// TIA Portal project "TestCase4_S1200_Zonder_Fouten " (V18)

(* hardware
DEVICE "S7-1200 station_1"  S7-1200 Station
   slot 0: "Rack_0"  S7-1200 Rack  Rack  V1.0
   slot 1: "PLC_1"  CPU 1212C DC/DC/DC  6ES7 212-1AE40-0XB0  V4.6
*)

// ===== PLC "PLC_1"  CPU 1212C DC/DC/DC =====

VAR_GLOBAL   // PLC tag table "Default tag table"
   "sensor1" AT %I0.0 : Bool;
   "lampA" AT %Q0.0 : Bool;
   "lampB" AT %Q0.1 : Bool;
   "Tag_1" AT %M101.0 : Bool;
   "Tag_2" AT %M100.0 : Bool;
   "Tag_4" AT %M100.1 : Bool;
   "Tag_5" AT %M100.2 : Bool;
   "sensor2" AT %I0.1 : Bool;
   "sensor3" AT %I0.2 : Bool;
   "Tag_6" AT %M103.0 : Bool;
   "Tag_7" AT %M102.0 : Bool;
END_VAR

DATA_BLOCK "Data_block_1"   // DB1
{ S7_Optimized_Access := 'FALSE' }
VERSION : 0.1
   VAR
      sensor1 : Bool;
      sensor2 : Bool;
      sensor3 : Bool;
   END_VAR
BEGIN
END_DATA_BLOCK

DATA_BLOCK "Data_block_2"   // DB2
{ S7_Optimized_Access := 'FALSE' }
VERSION : 0.1
   VAR
      lampA : Bool;
      lampB : Bool;
   END_VAR
BEGIN
END_DATA_BLOCK

FUNCTION "State0" : Void   // FC1, FBD
{ S7_Optimized_Access := 'TRUE' }
VERSION : 0.1
BEGIN

REGION Network 1
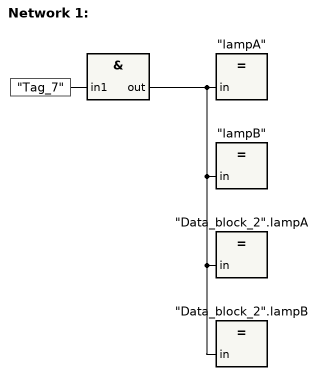
   "lampA" := "Tag_7";
   "lampB" := "Tag_7";
   "Data_block_2".lampA := "Tag_7";
   "Data_block_2".lampB := "Tag_7";
END_REGION
END_FUNCTION

FUNCTION "State1" : Void   // FC2, FBD
{ S7_Optimized_Access := 'TRUE' }
VERSION : 0.1
BEGIN

REGION Network 1
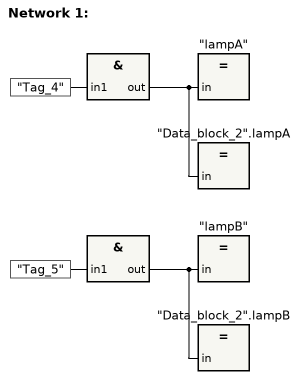
   "lampA" := "Tag_4";
   "Data_block_2".lampA := "Tag_4";
   "lampB" := "Tag_5";
   "Data_block_2".lampB := "Tag_5";
END_REGION
END_FUNCTION

FUNCTION "State2" : Void   // FC3, FBD
{ S7_Optimized_Access := 'TRUE' }
VERSION : 0.1
BEGIN

REGION Network 1
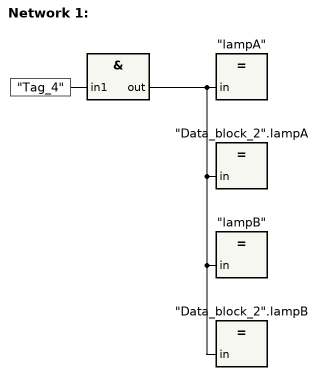
   "lampA" := "Tag_4";
   "Data_block_2".lampA := "Tag_4";
   "lampB" := "Tag_4";
   "Data_block_2".lampB := "Tag_4";
END_REGION
END_FUNCTION

ORGANIZATION_BLOCK "Main"   // OB1, FBD, ProgramCycle
TITLE = "Main Program Sweep (Cycle)"
{ S7_Optimized_Access := 'TRUE' }
VERSION : 0.1
   VAR_INPUT
      Initial_Call : Bool;   // Initial call of this OB
      Remanence : Bool;   // =True, if remanent data are available
   END_VAR
BEGIN

REGION Network 1
   // Initialize Merkers (M100.0 = 1 cycle true, M100.1 always 1 and M100.2 always 0).
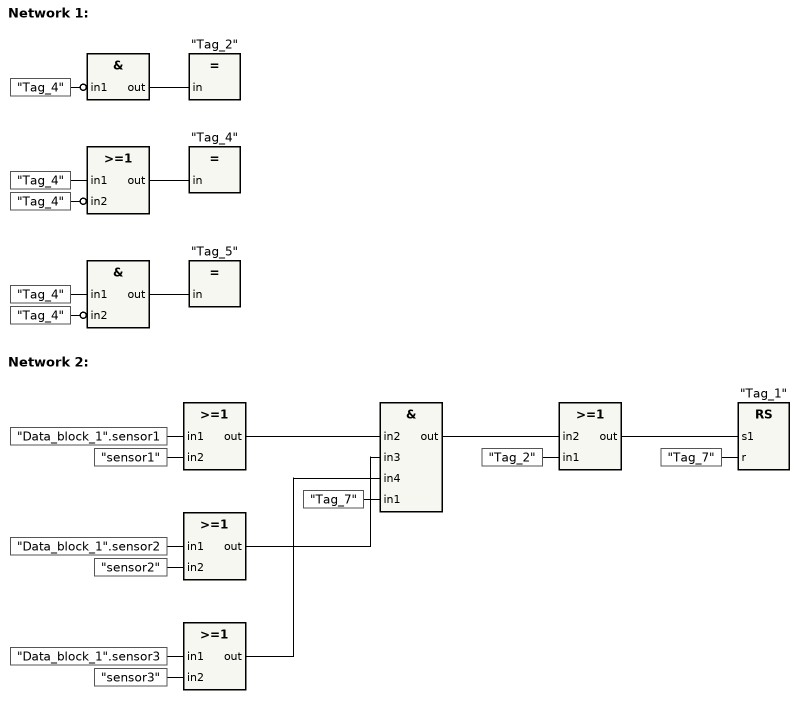
   "Tag_2" := NOT "Tag_4";
   "Tag_4" := "Tag_4" OR NOT "Tag_4";
   "Tag_5" := "Tag_4" AND NOT "Tag_4";
END_REGION

REGION Network 2
   // State 0
   IF "Tag_7" THEN
       "Tag_1" := FALSE;   // RS flip-flop
   END_IF;
   IF (("Data_block_1".sensor1 OR "sensor1") AND ("Data_block_1".sensor2 OR "sensor2") AND ("Data_block_1".sensor3 OR "sensor3") AND "Tag_7") OR "Tag_2" THEN
       "Tag_1" := TRUE;
   END_IF;
END_REGION

REGION Network 3
   // State 1
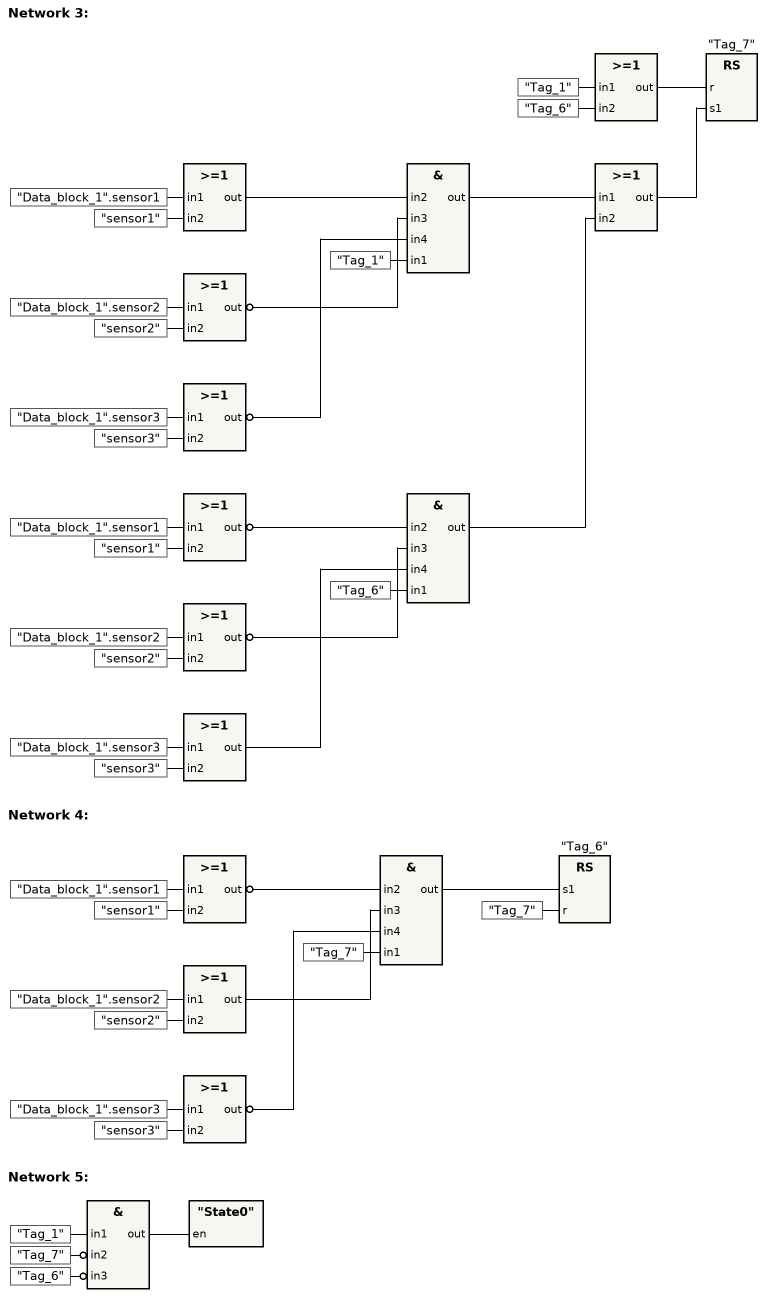
   IF "Tag_1" OR "Tag_6" THEN
       "Tag_7" := FALSE;   // RS flip-flop
   END_IF;
   IF (("Data_block_1".sensor1 OR "sensor1") AND NOT ("Data_block_1".sensor2 OR "sensor2") AND NOT ("Data_block_1".sensor3 OR "sensor3") AND "Tag_1") OR (NOT ("Data_block_1".sensor1 OR "sensor1") AND NOT ("Data_block_1".sensor2 OR "sensor2") AND ("Data_block_1".sensor3 OR "sensor3") AND "Tag_6") THEN
       "Tag_7" := TRUE;
   END_IF;
END_REGION

REGION Network 4
   // State 2
   IF "Tag_7" THEN
       "Tag_6" := FALSE;   // RS flip-flop
   END_IF;
   IF NOT ("Data_block_1".sensor1 OR "sensor1") AND ("Data_block_1".sensor2 OR "sensor2") AND NOT ("Data_block_1".sensor3 OR "sensor3") AND "Tag_7" THEN
       "Tag_6" := TRUE;
   END_IF;
END_REGION

REGION Network 5
   // Activate the outputs
   IF "Tag_1" AND NOT "Tag_7" AND NOT "Tag_6" THEN "State0"(); END_IF;
END_REGION

REGION Network 6
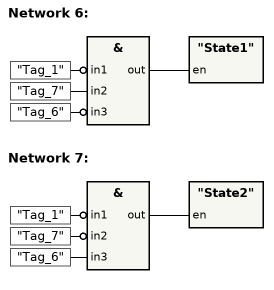
   IF NOT "Tag_1" AND "Tag_7" AND NOT "Tag_6" THEN "State1"(); END_IF;
END_REGION

REGION Network 7
   IF NOT "Tag_1" AND NOT "Tag_7" AND "Tag_6" THEN "State2"(); END_IF;
END_REGION
END_ORGANIZATION_BLOCK